Omron Sysmac Studio project SPA_P4 (Sysmac Studio 1.23.0.14, StandardProject)

# Controller new_Controller_0: NX1P2-1040DT1 version 1.18
Task PrimaryTask (priority 4, period or condition 2000): Programa0

PROGRAM Programa0
VAR
    valor1 : REAL;
    valor2 : REAL;
    valor3 : REAL;
    activacio : BOOL;
    calcul_ok : BOOL;
    resultat : REAL;
    dato_final : REAL;
END_VAR

(* Section MAIN: ladder, written here as Structured Text *)

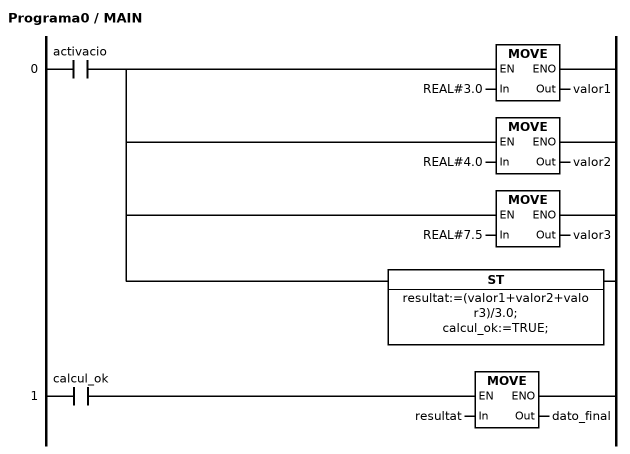
(* Rung 0 *)
IF activacio THEN
    valor1 := REAL#3.0;
    valor2 := REAL#4.0;
    valor3 := REAL#7.5;
END_IF;
IF activacio THEN
    resultat:=(valor1+valor2+valor3)/3.0;
    calcul_ok:=TRUE;
END_IF;
(* Rung 1 *)
IF calcul_ok THEN dato_final := resultat; END_IF;
END_PROGRAM